PROGRAM MAIN
VAR
END_VAR

FBD();

END_PROGRAM

(* stored: Version 1.1.0.1, ProductVersion 3.1.4024.12
   POU MAIN: Id {cf2a7ac2-c922-425a-abdf-6ff004b3acb3}, SpecialFunc None *)
